// TIA Portal project "btvn_tuan2" (V14)

(* hardware
DEVICE "S7-1200 station_1"  S7-1200 Station
   slot 0: "Rack_0"  S7-1200 Rack  Rack  V1.0
   slot 1: "PLC_1"  CPU 1214C DC/DC/DC  6ES7 214-1AG40-0XB0  V4.2
*)

// ===== PLC "PLC_1"  CPU 1214C DC/DC/DC =====

VAR_GLOBAL   // PLC tag table "Default tag table"
   "gia tri cam bien" AT %IW64 : Word;
   "tmp" AT %MD10 : Real;
   "nhiet do" AT %MD4 : Real;
   "Start/Stop" AT %M0.0 : Bool;
   "qua nhiet" AT %M0.1 : Bool;
   "motor khuay" AT %M0.2 : Bool;
   "phase1" AT %M0.3 : Bool;
   "phase2" AT %M0.4 : Bool;
   "up" AT %M0.5 : Bool;
   "vd" AT %M0.6 : Bool;
END_VAR

// folder: System blocks/Program resources

DATA_BLOCK "IEC_Timer_0_DB"   // DB1
{ S7_Optimized_Access := 'TRUE' }
AUTHOR : Simatic
FAMILY : IEC
NAME : IEC_TMR
VERSION : 1.0
// stored: InstanceOfName IEC_TIMER
"IEC_TIMER"
BEGIN
END_DATA_BLOCK

DATA_BLOCK "IEC_Timer_0_DB_1"   // DB2
{ S7_Optimized_Access := 'TRUE' }
AUTHOR : Simatic
FAMILY : IEC
NAME : IEC_TMR
VERSION : 1.0
// stored: InstanceOfName IEC_TIMER
"IEC_TIMER"
BEGIN
END_DATA_BLOCK

// folder: (top level)

ORGANIZATION_BLOCK "Main"   // OB1, LAD, ProgramCycle
TITLE = "Main Program Sweep (Cycle)"
{ S7_Optimized_Access := 'TRUE' }
VERSION : 0.1
   VAR_INPUT
      Initial_Call : Bool;   // Initial call of this OB
      Remanence : Bool;   // =True, if remanent data are available
   END_VAR
   VAR_TEMP   // added for the SCL form of the ladder/FBD networks
      _w1 : Bool;
   END_VAR
BEGIN

REGION Network 1: lay nhiet do
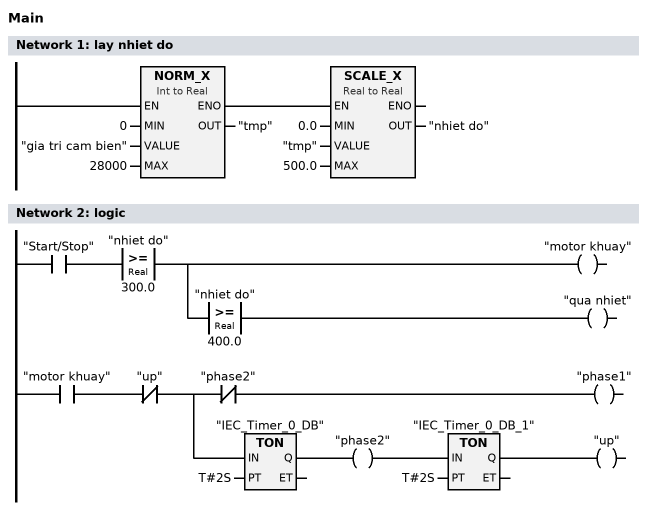
   RUNG wire#powerrail
      { S7_Templates := "[SrcType := Int, DestType := Real]" } Normalize(min := 0, value := "gia tri cam bien", max := 28000, out => "tmp")
      { S7_Templates := "[SrcType := Real, DestType := Real]" } Scale(min := 0.0, value := "tmp", max := 500.0, out => "nhiet do")
   END_RUNG
   // the same network as SCL:
   "tmp" := NORM_X(MIN := 0, VALUE := "gia tri cam bien", MAX := 28000);
   "nhiet do" := SCALE_X(MIN := 0.0, VALUE := "tmp", MAX := 500.0);
END_REGION

REGION Network 2: logic
   "motor khuay" := "Start/Stop" AND ("nhiet do" >= 300.0);
   "qua nhiet" := "motor khuay" AND ("nhiet do" >= 400.0);
   #_w1 := "motor khuay" AND NOT "up";
   "phase1" := #_w1 AND NOT "phase2";
   "IEC_Timer_0_DB".TON(IN := #_w1, PT := T#2S);
   "phase2" := "IEC_Timer_0_DB".Q;
   "IEC_Timer_0_DB_1".TON(IN := "IEC_Timer_0_DB".Q, PT := T#2S);
   "up" := "IEC_Timer_0_DB_1".Q;
END_REGION
END_ORGANIZATION_BLOCK